(* CODESYS project CodesysEEN150_Lab_cylinders.export

Project tree, tasks and I/O mapping:
  Device : CODESYS Control Win V3, 3S - Smart Software Solutions GmbH, version 3.5.16.0
    application Application
      libraries: Standard, * (System); CmpBitmapPool, * (System); Util, * (System)
      task MainTask (cyclic, interval 5 ms, priority 1) calls cylinder_control_SFC
      task simulation (cyclic, interval t#20ms, priority 1) calls sim_logic
      task VISU_TASK (cyclic, interval 10 ms, priority 31) calls VisuElems.Visu_Prg
      control/
        function block CylinderFB [LD]
        function block CylinderFB_1 [LD]
        program CylinderFB_old [FBD]
        program cylinder_control_SFC [LD]
        program cylinder_ctrl [LD]
        program cylinder_ctrl_1 [LD]
        function block LampCTRL [SFC]
        function block Sequence [SFC]
      simulation/
        function block cylSimulation [ST]
        program sim_logic [LD]
      global variables IO
      image pool ImagePool
      visualisation Cylinders
  5ce3da45-db07-42e7-a21c-a00fff4ed8f6|C:\Users\ryytt\OneDrive\Skrivbord\examensarbete\bakgrund.png
  5ce3da45-db07-42e7-a21c-a00fff4ed8f6|C:\Users\ryytt\OneDrive\Skrivbord\examensarbete\bakgrundv2.png
*)

// Device/Application/IO
VAR_GLOBAL
	ixStart: BOOL; // the start switch and the button
 	ixStop: BOOL;  // the stop switch and the button
	ixReset: BOOL; // the reset switch
	ixB1: BOOL; // button B1
	ixB2: BOOL; // button B2
	ixIN10: BOOL; // the IN10 switch
	ixIN11: BOOL; // the IN11 switch
	ixCylinder1In: BOOL; // a sensor if cylinder 1 is in
	ixCylinder1Out: BOOL; // a sensor if cylinder 1 is in
	ixCylinder2In: BOOL; // a sensor if cylinder 1 is in
	ixCylinder2Out: BOOL; // a sensor if cylinder 1 is in
	ixCylinder3In: BOOL; // a sensor if cylinder 1 is in
	ixCylinder3Out: BOOL; // a sensor if cylinder 1 is in	
	ixEmergencyStop: BOOL := TRUE; // the emergency stop. If false, it is active

	qxLamp1: BOOL; // to control L1
	qxLamp2: BOOL; // to control L2
	qxLamp3: BOOL; // to ontorl L3
	qxLamp4: BOOL; // to control L4
	qxCylinder1: BOOL; // to extend cylinder 1
	qxCylinder2: BOOL; // to extend cylinder 2
	qxCylinder3: BOOL; // to extend cylinder 3
END_VAR

// Device/Application/control/cylinder_control_SFC
PROGRAM cylinder_control_SFC
VAR
	cylinder1: CylinderFB;
	cylinder2: CylinderFB;
	cylinder3: CylinderFB;
	CylinderFB_0: CylinderFB;
	start_cyl_2: BOOL := FALSE;
	init: BOOL := TRUE;
	starting: BOOL;
	cyl_1_out: BOOL ;
	cyl_1_done: BOOL := FALSE;
	cyl_1_retract: BOOL;
	sequence1: Sequence;
END_VAR
VAR // added by the converter: edge detectors and wires of the graphical bodies
    _rt1, _rt2 : R_TRIG;
END_VAR

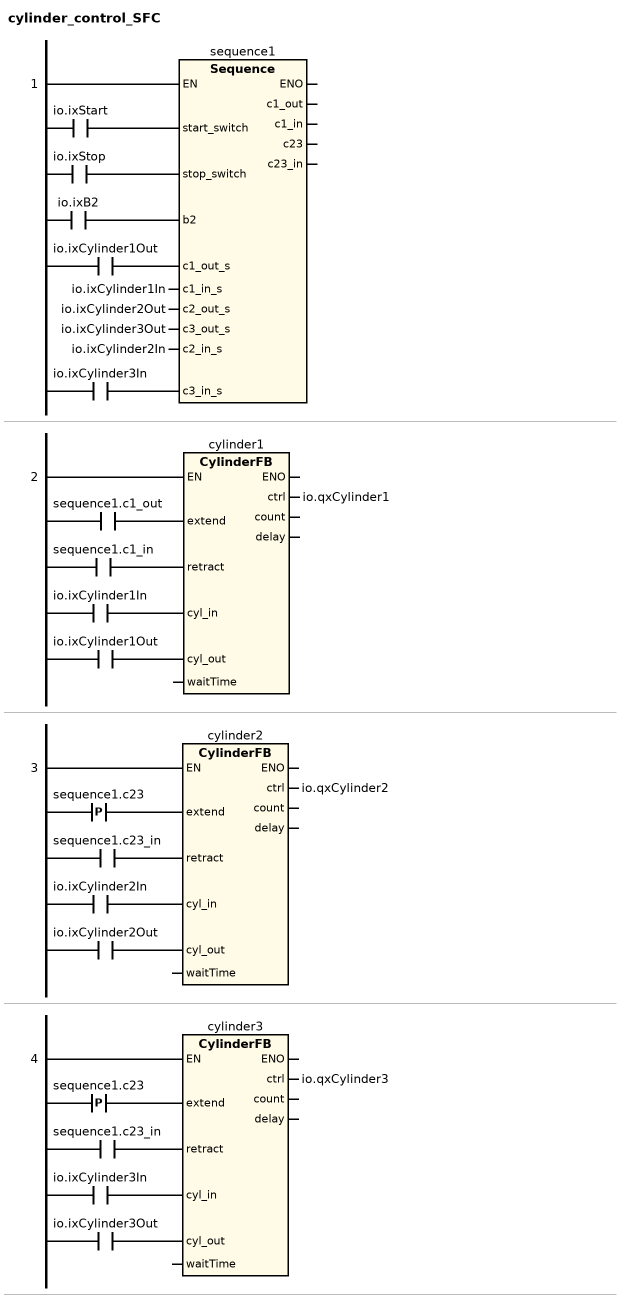
// NETWORK 1
sequence1(
    start_switch := io.ixStart,
    stop_switch := io.ixStop,
    b2 := io.ixB2,
    c1_out_s := io.ixCylinder1Out,
    c1_in_s := io.ixCylinder1In,
    c2_out_s := io.ixCylinder2Out,
    c3_out_s := io.ixCylinder3Out,
    c2_in_s := io.ixCylinder2In,
    c3_in_s := io.ixCylinder3In); // Sequence

// NETWORK 2
cylinder1(
    extend := sequence1.c1_out,
    retract := sequence1.c1_in,
    cyl_in := io.ixCylinder1In,
    cyl_out := io.ixCylinder1Out,
    ctrl => io.qxCylinder1); // CylinderFB

// NETWORK 3
_rt1(CLK := sequence1.c23);
cylinder2(
    extend := _rt1.Q,
    retract := sequence1.c23_in,
    cyl_in := io.ixCylinder2In,
    cyl_out := io.ixCylinder2Out,
    ctrl => io.qxCylinder2); // CylinderFB

// NETWORK 4
_rt2(CLK := sequence1.c23);
cylinder3(
    extend := _rt2.Q,
    retract := sequence1.c23_in,
    cyl_in := io.ixCylinder3In,
    cyl_out := io.ixCylinder3Out,
    ctrl => io.qxCylinder3); // CylinderFB

END_PROGRAM

// Device/Application/control/Sequence
FUNCTION_BLOCK Sequence
VAR_INPUT
	start_switch: BOOL;
	stop_switch: BOOL;
	b2:BOOL;
	c1_out_s:BOOL;
	c1_in_s: BOOL;
	c2_out_s: BOOL;
	c3_out_s: BOOL;
	c2_in_s: BOOL;
	c3_in_s: BOOL;
END_VAR
VAR_OUTPUT
	c1_out:BOOL;
	c1_in:BOOL;
	c23:BOOL;
	c23_in: BOOL;
END_VAR
VAR
END_VAR

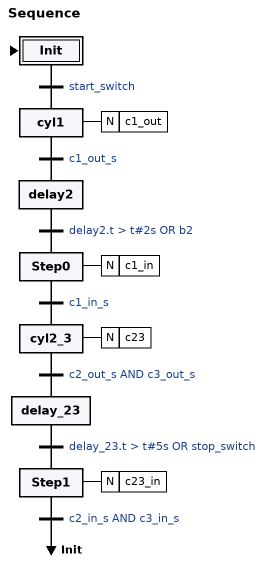
INITIAL_STEP Init:
END_STEP
TRANSITION FROM Init TO cyl1
    := start_switch;
END_TRANSITION
STEP cyl1:
    c1_out(N);
END_STEP
TRANSITION FROM cyl1 TO delay2
    := c1_out_s;
END_TRANSITION
STEP delay2:
END_STEP
TRANSITION FROM delay2 TO Step0
    := delay2.t > t#2s OR b2;
END_TRANSITION
STEP Step0:
    c1_in(N);
END_STEP
TRANSITION FROM Step0 TO cyl2_3
    := c1_in_s;
END_TRANSITION
STEP cyl2_3:
    c23(N);
END_STEP
TRANSITION FROM cyl2_3 TO delay_23
    := c2_out_s AND c3_out_s;
END_TRANSITION
STEP delay_23:
END_STEP
TRANSITION FROM delay_23 TO Step1
    := delay_23.t > t#5s OR stop_switch;
END_TRANSITION
STEP Step1:
    c23_in(N);
END_STEP
TRANSITION FROM Step1 TO Init
    := c2_in_s AND c3_in_s;
END_TRANSITION

END_FUNCTION_BLOCK

// Device/Application/control/CylinderFB
FUNCTION_BLOCK CylinderFB
VAR_INPUT
	extend: BOOL;
	retract: BOOL;
	cyl_in: BOOL;
	cyl_out: BOOL;
	waitTime: TIME;
END_VAR
VAR_OUTPUT
	ctrl: BOOL;
	count: INT := 0;
	delay: TIME := T#0S;
END_VAR
VAR
	stop: BOOL := FALSE;
	timer: TON;
END_VAR
VAR // added by the converter: edge detectors and wires of the graphical bodies
    _rt1, _rt2 : R_TRIG;
END_VAR

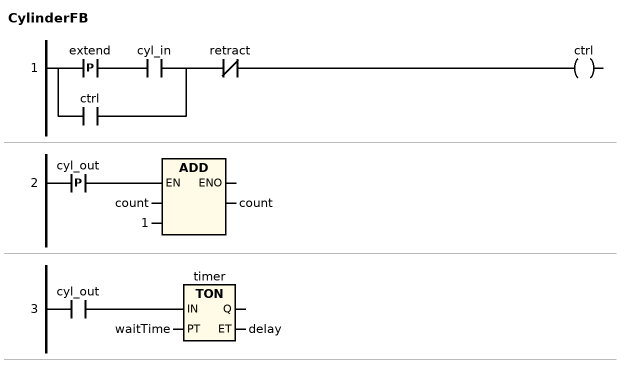
// NETWORK 1
_rt1(CLK := extend);
ctrl := (_rt1.Q AND cyl_in OR ctrl) AND NOT retract;

// NETWORK 2
_rt2(CLK := cyl_out);
IF _rt2.Q THEN count := count + 1; END_IF

// NETWORK 3
timer(IN := cyl_out, PT := waitTime, ET => delay); // TON

END_FUNCTION_BLOCK

// Device/Application/simulation/sim_logic
PROGRAM sim_logic
VAR
	cyl1: cylSimulation;
	donotuse_cyl1_pos: INT;
	cyl2: cylSimulation;
	cyl3: cylSimulation;
	donotuse_cyl2_pos: INT;
	donotuse_cyl3_pos: INT;
END_VAR

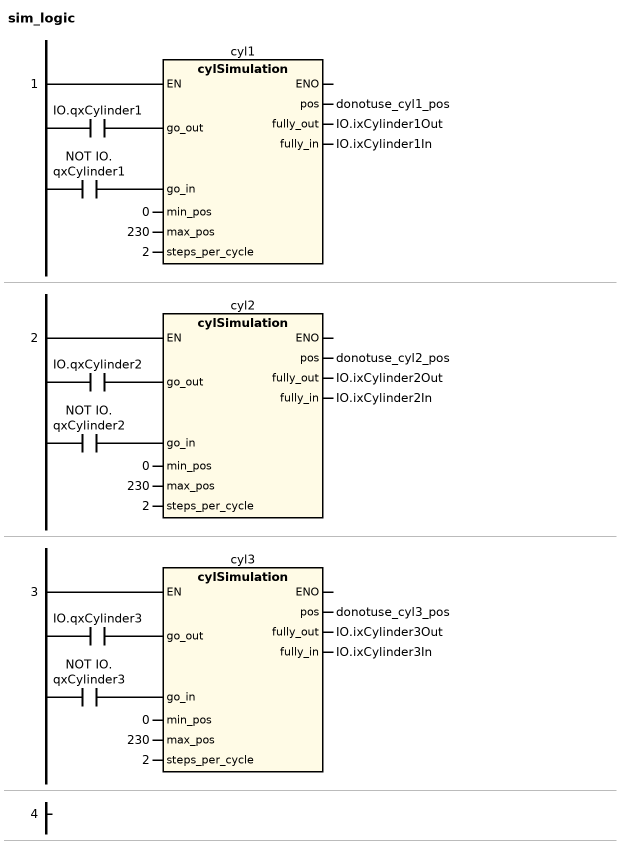
// NETWORK 1
cyl1(
    go_out := IO.qxCylinder1,
    go_in := NOT IO.qxCylinder1,
    min_pos := 0,
    max_pos := 230,
    steps_per_cycle := 2,
    pos => donotuse_cyl1_pos,
    fully_out => IO.ixCylinder1Out,
    fully_in => IO.ixCylinder1In); // cylSimulation

// NETWORK 2
cyl2(
    go_out := IO.qxCylinder2,
    go_in := NOT IO.qxCylinder2,
    min_pos := 0,
    max_pos := 230,
    steps_per_cycle := 2,
    pos => donotuse_cyl2_pos,
    fully_out => IO.ixCylinder2Out,
    fully_in => IO.ixCylinder2In); // cylSimulation

// NETWORK 3
cyl3(
    go_out := IO.qxCylinder3,
    go_in := NOT IO.qxCylinder3,
    min_pos := 0,
    max_pos := 230,
    steps_per_cycle := 2,
    pos => donotuse_cyl3_pos,
    fully_out => IO.ixCylinder3Out,
    fully_in => IO.ixCylinder3In); // cylSimulation

// NETWORK 4

END_PROGRAM

// Device/Application/simulation/cylSimulation
FUNCTION_BLOCK cylSimulation
VAR_INPUT
	go_out: BOOL;
	go_in: BOOL;
	min_pos: INT;
	max_pos: INT;
	steps_per_cycle: INT;
END_VAR
VAR_OUTPUT
	pos: INT;
	fully_out: BOOL;
	fully_in: BOOL;
END_VAR
VAR
END_VAR


IF go_out AND NOT go_in THEN
	pos := pos + steps_per_cycle;
END_IF
IF go_in AND NOT go_out THEN
	pos := pos - steps_per_cycle;
END_IF

pos := LIMIT(min_pos, pos, max_pos);

fully_in := pos = min_pos;
fully_out := pos = max_pos;

END_FUNCTION_BLOCK

// Device/Application/control/CylinderFB_1
FUNCTION_BLOCK CylinderFB_1
VAR_INPUT
	extend: BOOL;
	retract: BOOL;
	cyl_in: BOOL;
	cyl_out: BOOL;
	waitTime: TIME;
END_VAR
VAR_OUTPUT
	ctrl: BOOL;
	count: INT := 0;
	delay: TIME := T#0S;
END_VAR
VAR
	stop: BOOL := FALSE;
	timer: TON;
END_VAR
VAR // added by the converter: edge detectors and wires of the graphical bodies
    _rt1, _rt2 : R_TRIG;
END_VAR

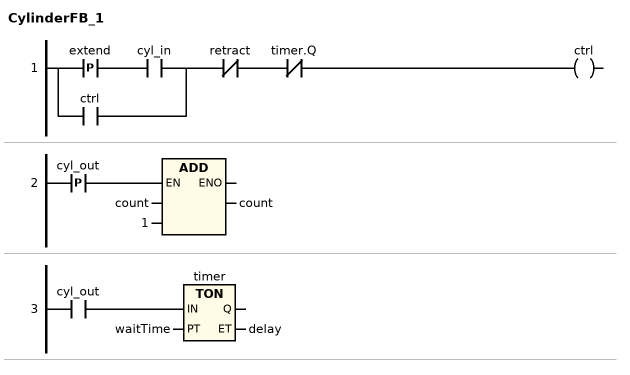
// NETWORK 1
_rt1(CLK := extend);
ctrl := (_rt1.Q AND cyl_in OR ctrl) AND NOT retract AND NOT timer.Q;

// NETWORK 2
_rt2(CLK := cyl_out);
IF _rt2.Q THEN count := count + 1; END_IF

// NETWORK 3
timer(IN := cyl_out, PT := waitTime, ET => delay); // TON

END_FUNCTION_BLOCK

// Device/Application/control/CylinderFB_old
PROGRAM CylinderFB_old
VAR_INPUT
	extend: BOOL;
	retract: BOOL;
	cyl_in: BOOL;
	cyl_out: BOOL;
END_VAR
VAR_OUTPUT
	ctrl: BOOL;
	count: INT := 0;
END_VAR
VAR
END_VAR
VAR // added by the converter: edge detectors and wires of the graphical bodies
    _rt1 : R_TRIG;
END_VAR

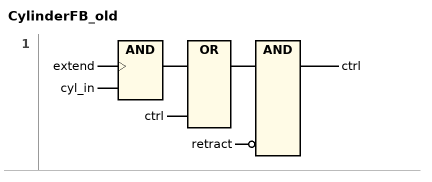
// NETWORK 1
_rt1(CLK := extend);
ctrl := (_rt1.Q AND cyl_in OR ctrl) AND NOT retract;

END_PROGRAM

// Device/Application/control/cylinder_ctrl
PROGRAM cylinder_ctrl
VAR
	cylinder1: CylinderFB;
	cylinder2: CylinderFB;
	cylinder3: CylinderFB;
	CylinderFB_0: CylinderFB;
	start_cyl_2: BOOL := FALSE;
	init: BOOL := TRUE;
	starting: BOOL;
	cyl_1_out: BOOL ;
	cyl_1_done: BOOL := FALSE;
END_VAR
VAR // added by the converter: edge detectors and wires of the graphical bodies
    _rt1, _rt2 : R_TRIG;
    _w1, _w2 : BOOL;
END_VAR

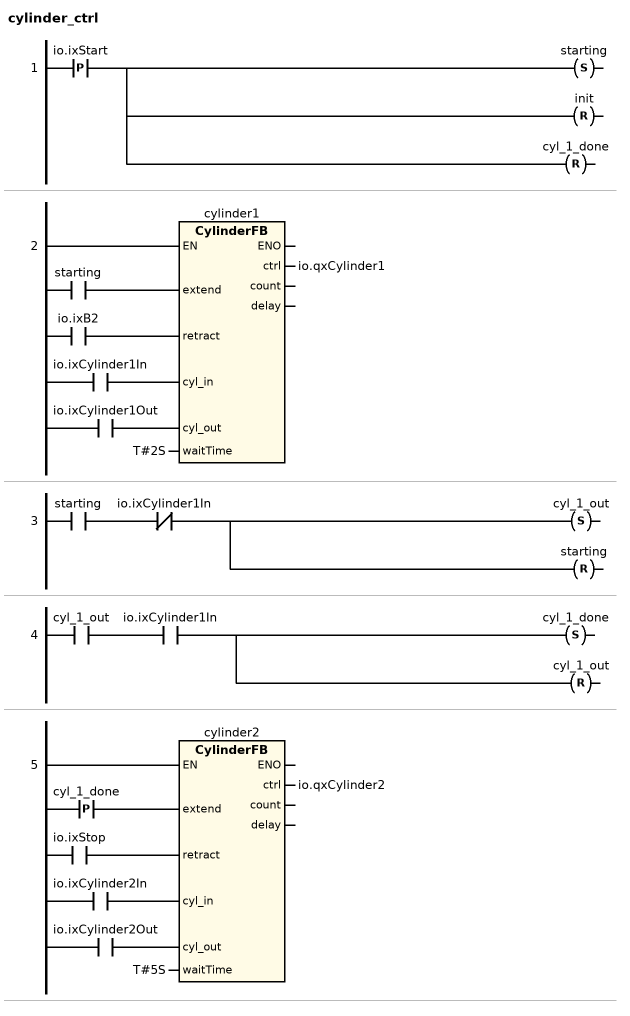
// NETWORK 1
_rt1(CLK := io.ixStart);
starting S= _rt1.Q;
init R= _rt1.Q;
cyl_1_done R= _rt1.Q;

// NETWORK 2
cylinder1(
    extend := starting,
    retract := io.ixB2,
    cyl_in := io.ixCylinder1In,
    cyl_out := io.ixCylinder1Out,
    waitTime := T#2S,
    ctrl => io.qxCylinder1); // CylinderFB

// NETWORK 3
_w1 := starting AND NOT io.ixCylinder1In;
cyl_1_out S= _w1;
starting R= _w1;

// NETWORK 4
_w2 := cyl_1_out AND io.ixCylinder1In;
cyl_1_done S= _w2;
cyl_1_out R= _w2;

// NETWORK 5
_rt2(CLK := cyl_1_done);
cylinder2(
    extend := _rt2.Q,
    retract := io.ixStop,
    cyl_in := io.ixCylinder2In,
    cyl_out := io.ixCylinder2Out,
    waitTime := T#5S,
    ctrl => io.qxCylinder2); // CylinderFB

END_PROGRAM

// Device/Application/control/cylinder_ctrl_1
PROGRAM cylinder_ctrl_1
VAR
	cylinder1: CylinderFB;
	cylinder2: CylinderFB;
	cylinder3: CylinderFB;
	CylinderFB_0: CylinderFB;
	start_cyl_2: BOOL := FALSE;
	init: BOOL := TRUE;
	starting: BOOL;
	cyl_1_out: BOOL ;
	cyl_1_done: BOOL := FALSE;
	lamp_testing: LampCTRL;
END_VAR

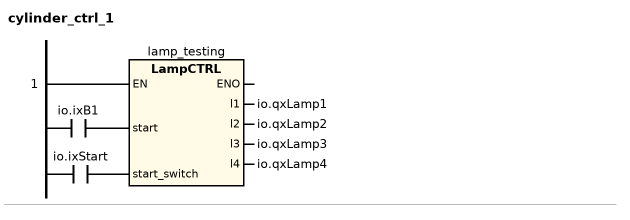
// NETWORK 1
lamp_testing(
    start := io.ixB1,
    start_switch := io.ixStart,
    l1 => io.qxLamp1,
    l2 => io.qxLamp2,
    l3 => io.qxLamp3,
    l4 => io.qxLamp4); // LampCTRL

END_PROGRAM

// Device/Application/control/LampCTRL
FUNCTION_BLOCK LampCTRL
VAR_INPUT
	 start: BOOL;
	 start_switch: BOOL;
END_VAR
VAR_OUTPUT
	l1: BOOL;
	l2: BOOL;
	l3: BOOL;
	l4: BOOL;
END_VAR
VAR
END_VAR

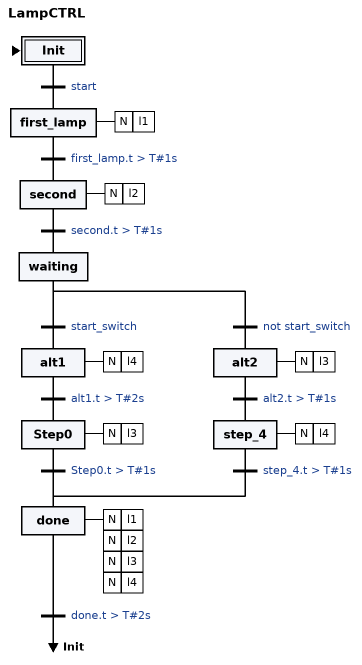
INITIAL_STEP Init:
END_STEP
TRANSITION FROM Init TO first_lamp
    := start;
END_TRANSITION
STEP first_lamp:
    l1(N);
END_STEP
TRANSITION FROM first_lamp TO second
    := first_lamp.t > T#1s;
END_TRANSITION
STEP second:
    l2(N);
END_STEP
TRANSITION FROM second TO waiting
    := second.t > T#1s;
END_TRANSITION
STEP waiting:
END_STEP
TRANSITION FROM waiting TO alt1
    := start_switch;
END_TRANSITION
STEP alt1:
    l4(N);
END_STEP
TRANSITION FROM alt1 TO Step0
    := alt1.t > T#2s;
END_TRANSITION
STEP Step0:
    l3(N);
END_STEP
TRANSITION FROM Step0 TO done
    := Step0.t > T#1s;
END_TRANSITION
TRANSITION FROM waiting TO alt2
    := not start_switch;
END_TRANSITION
STEP alt2:
    l3(N);
END_STEP
TRANSITION FROM alt2 TO step_4
    := alt2.t > T#1s;
END_TRANSITION
STEP step_4:
    l4(N);
END_STEP
TRANSITION FROM step_4 TO done
    := step_4.t > T#1s;
END_TRANSITION
STEP done:
    l1(N);
    l2(N);
    l3(N);
    l4(N);
END_STEP
TRANSITION FROM done TO Init
    := done.t > T#2s;
END_TRANSITION

END_FUNCTION_BLOCK

// Device/Application/Cylinders
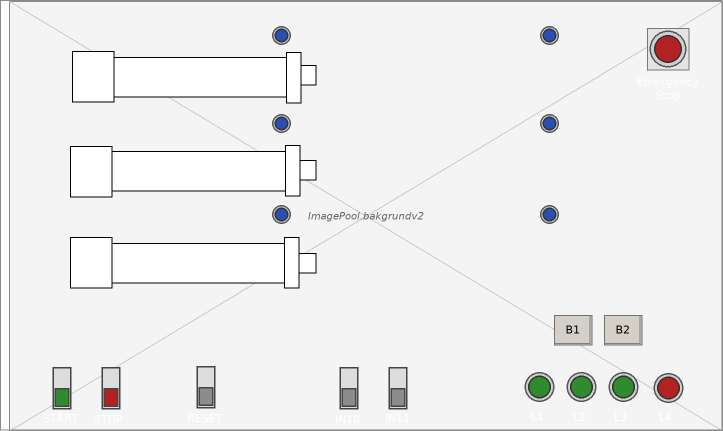
VISUALIZATION Cylinders  // 723x431
    Image (9,1 714x430), image: ImagePool.bakgrundv2
    Rectangle (286,253 30x20)
        p874137650: sim_logic.donotuse_cyl3_pos
    Rectangle (286,160 30x20)
        p874137650: sim_logic.donotuse_cyl2_pos
    Lamp1 (522,370 35x34), tooltip "L1", variable: qxLamp1, style: Lamp-Lamp1-Green
    Lamp1 (564,370 35x34), tooltip "L2", variable: qxLamp2, style: Lamp-Lamp1-Green
    Lamp1 (606,370 35x34), tooltip "L3", variable: qxLamp3, style: Lamp-Lamp1-Green
    Lamp1 (651,371 35x34), tooltip "L4", variable: qxLamp4, style: Lamp-Lamp1-Red
    DipSwitch (41,366 42x44), variable: ixStart, behaviour: TOGGLE, style: Switch-DipSwitch-Green
    DipSwitch (90,366 42x44), variable: ixStop, behaviour: TOGGLE, style: Switch-DipSwitch-Red
    DipSwitch (185,365 42x44), tooltip "RESET", variable: ixReset, behaviour: TOGGLE, style: Switch-DipSwitch-Gray
    DipSwitch (328,366 42x44), variable: ixIN10, behaviour: TOGGLE, style: Switch-DipSwitch-Gray
    DipSwitch (377,366 42x44), variable: ixIN11, behaviour: TOGGLE, style: Switch-DipSwitch-Gray
    Label (16,409 89x19), "START"
    Label (64,410 89x19), "STOP"
    Label (160,409 89x19), "RESET"
    Label (303,410 89x19), "IN10"
    Label (353,409 89x19), "IN11"
    Label (493,407 89x19), "L1"
    Label (535,408 89x19), "L2"
    Label (576,408 89x19), "L3"
    Label (621,408 89x19), "L4"
    Rectangle (286,65 30x20)
        p874137650: sim_logic.donotuse_cyl1_pos
    Rectangle (101,57 193x40)
    Rectangle (99,151 193x40)
    Rectangle (102,243 193x40)
    RoundedRectangle (70,237 42x51), "CYL3"
    RoundedRectangle (70,146 42x51), "CYL2"
    RoundedRectangle (72,51 42x51), "CYL1"
    RoundedRectangle (286,52 15x51)
    RoundedRectangle (285,145 15x51)
    RoundedRectangle (284,237 15x51)
    Lamp1 (271,25 21x21), variable: ixCylinder1In, style: Lamp-Lamp1-Blue
    Lamp1 (539,25 21x21), variable: ixCylinder1Out, style: Lamp-Lamp1-Blue
    Lamp1 (271,113 21x21), variable: ixCylinder2In, style: Lamp-Lamp1-Blue
    Lamp1 (539,113 21x21), variable: ixCylinder2Out, style: Lamp-Lamp1-Blue
    Lamp1 (271,204 21x21), variable: ixCylinder3In, style: Lamp-Lamp1-Blue
    Lamp1 (539,204 21x21), variable: ixCylinder3Out, style: Lamp-Lamp1-Blue
    PushSwitch (647,27 42x44), variable: ixEmergencyStop, behaviour: TOGGLE, style: Switch-PushSwitch-Red
    Label (623,72 90x33), "Emergency Stop"
    Button (554,315 38x30), "B1"
        tap ixB1
    Button (604,315 38x30), "B2"
        tap ixB2
END_VISUALIZATION
